(*

.. <legal notes>

legal notes
=================
| SPDX-FileCopyrightText: © 2026 Oleksandr Tiutyk <trofimich@gmail.com>
| SPDX-License-Identifier: LGPL-3.0-only
| For details check: LGPL-3.0-only_

.. _LGPL-3.0-only: https://www.gnu.org/licenses/lgpl-3.0.en.html

.. </legal notes>

*)

TYPE HMI_AUTOMATION_CONTROLLER_BASE_COMMANDS :
STRUCT
	Enable : BOOL;
	Disable : BOOL;
	
	Reset : BOOL;	
END_STRUCT
END_TYPE

(* stored: Version 1.1.0.1
   DUT HMI_AUTOMATION_CONTROLLER_BASE_COMMANDS: Id {1590423e-7120-451f-b462-35fc53b7d967} *)
